Fanuc KAREL source: ke00001.KL

PROGRAM KE00001
%NOLOCKGROUP
%ENVIRONMENT REGOPE
VAR
I:INTEGER;S : STRING[80];STATUS:INTEGER
BEGIN
--
--
I=1
GET_PREG_CMT(I,S,STATUS)
END KE00001
